FUNCTION_BLOCK EL3061
VAR
	_io : EL3xx1_Data;
	{attribute addProperty Name "WcState"}
	_wcState : WcStateInputToggle;
	{attribute addProperty Name "Info data"}
	_infoData : InfoDataAds;
END_VAR

PROPERTY IO : REFERENCE TO EL3xx1_Data
GET
IO REF= _io;
END_GET
END_PROPERTY

PROPERTY WcState : REFERENCE TO WcStateInputToggle
GET
WcState REF= _wcState;
END_GET
END_PROPERTY

END_FUNCTION_BLOCK

(* stored: Version 1.1.0.1, ProductVersion 3.1.4024.9
   POU EL3061: Id {ac6d3b73-23f7-0914-1084-24204dccae69}, SpecialFunc None
   Property IO: Id {184fcff0-a6f3-0552-2eab-6173cc4085d3}
   Get Get: Id {d4f7c64a-a6ab-069f-3808-700b415063e0}
   Property WcState: Id {68670786-6f48-056f-152f-633d3514dccd}
   Get Get: Id {a8f3ce5d-a686-0a08-36ad-e63af865d36d} *)
